(* PLC project WEEE_PLCs, Sconosciuto Senza_nome 1 *)
(* stored: creationDateTime 2024-08-18T12:18:40, modificationDateTime 2025-04-19T20:38:53 *)

TYPE STATUSES : (SHUT, OK, DANGER);
END_TYPE

TYPE FUNCTIONALITIES : (CONTROLLER, SEPARATOR);
END_TYPE

TYPE PLATFORM : STRUCT
  ID : INT;
  SHUTTED : BOOL;
  PC : REAL;
  SETTING : SETTINGS;
  STATUS : STATUSES;
  DIRECTION : DIRECTIONS;
  MATERIAL : MATERIALS;
END_STRUCT;
END_TYPE

TYPE SETTINGS : (AUTO, MANUAL);
END_TYPE

TYPE DIRECTIONS : (FORWARD, BACKWARD);
END_TYPE

TYPE WEIGHTS : (L, M, H);
END_TYPE

TYPE MATERIALS : (STEEL, COPPER, GOLD, CLAY, STONE);
END_TYPE

TYPE SHREADER : STRUCT
  ID : INT;
  PC : REAL;
  SETTING : SETTINGS;
  STATUS : STATUSES;
  WEIGHT : WEIGHTS;
END_STRUCT;
END_TYPE

FUNCTION_BLOCK PLATFORM_FB
  VAR_INPUT
    SHUTTED_IN : BOOL;
    SETTING_IN : INT;
    STATUS_IN : INT;
    PLATFORM_IN : PLATFORM;
  END_VAR
  VAR_OUTPUT
    STATUS_OUT : INT;
    PLATFORM_OUT : PLATFORM;
  END_VAR

            (*PLATFORM REMOTE CONFIGURATION*)
CASE SETTING_IN OF
  0: PLATFORM_IN.SETTING := MANUAL;
  1: PLATFORM_IN.SETTING := AUTO;
END_CASE;

(*SET PC BASED ON STATUS*)
IF SHUTTED_IN THEN
  PLATFORM_OUT.PC := 0.0;
  RETURN;
ELSE
  PLATFORM_OUT.PC := 3.5;
END_IF;

(*SET STATUS TO DANGER IF SOMETHING IS NOT NORMAL*)
IF PLATFORM_IN.PC >= 10.0 THEN
  PLATFORM_OUT.STATUS := DANGER;
ELSE
  PLATFORM_OUT.STATUS := OK;
END_IF;

(*UPDATE STATUS FOR MODBUS*)
CASE PLATFORM_OUT.STATUS OF
  OK: STATUS_OUT := 0;
  DANGER: STATUS_OUT := 1;
END_CASE;




          
END_FUNCTION_BLOCK

PROGRAM ClensePlc
  VAR
    C_ID : INT := 4;
    C_SHUTTED : BOOL;
    C_PILOT_STATUS : INT;
    C_PILOT_FUNC : INT;
    C_PC_INT : INT;
    C_STATUS : STATUSES;
    C_FUNC : FUNCTIONALITIES := CONTROLLER;
    C_PC_REAL : REAL := 0.0;
    C_WASTE_FB : PLATFORM_FB;
    C_WASTE : PLATFORM;
    C_WASTE_ID : INT := 8;
    C_WASTE_PC : REAL := 0.0;
    C_WASTE_SETTING : INT;
    C_WASTE_STATUS : INT;
    C_WASTE_DIRECTION : INT;
    C_WASTE_MATERIAL : INT;
  END_VAR
  VAR_EXTERNAL
    DENSITIES : ARRAY[0..2] OF PLATFORM;
  END_VAR
  VAR
    C_DENS_H_FB : PLATFORM_FB;
  END_VAR
  VAR_EXTERNAL
    DENS_H : PLATFORM;
    DENS_H_ID : INT;
    DENS_H_PC : REAL;
    DENS_H_SETTING : INT;
    DENS_H_STATUS : INT;
    DENS_H_DIRECTION : INT;
    DENS_H_MATERIAL : INT;
  END_VAR
  VAR
    C_DENS_M_FB : PLATFORM_FB;
  END_VAR
  VAR_EXTERNAL
    DENS_M : PLATFORM;
    DENS_M_ID : INT;
    DENS_M_PC : REAL;
    DENS_M_SETTING : INT;
    DENS_M_STATUS : INT;
    DENS_M_DIRECTION : INT;
    DENS_M_MATERIAL : INT;
  END_VAR
  VAR
    C_DENS_L_FB : PLATFORM_FB;
  END_VAR
  VAR_EXTERNAL
    DENS_L : PLATFORM;
    DENS_L_ID : INT;
    DENS_L_PC : REAL;
    DENS_L_SETTING : INT;
    DENS_L_STATUS : INT;
    DENS_L_DIRECTION : INT;
    DENS_L_MATERIAL : INT;
  END_VAR

            (*Define logic to assign enum value when receiving a command through modbus*)


(*Make the changes needed inside the function
C_WASTE_FB(
     IN := C_WASTE,
     OUT => C_WASTE);
*)

(*Update the variables with the new ones*)
C_WASTE_PC := C_WASTE.PC;

(*Set C_STATUS based on remote input*)


(*logic for functionality status*)



          
END_PROGRAM

PROGRAM DensityPlc
  VAR
    D_ID AT %QW3 : INT := 3;
  END_VAR
  VAR
    D_PC : REAL := 0.0;
    D_STATUS : STATUSES;
    D_PILOT_STATUS : INT;
    D_FUNC : FUNCTIONALITIES := SEPARATOR;
    D_GRIST_FB : PLATFORM_FB;
    D_GRIST : PLATFORM;
    D_GRIST_ID : INT := 20;
    D_GRIST_PC : REAL := 0.0;
    D_GRIST_SETTING : INT;
    D_GRIST_STATUS : INT;
    D_GRIST_DIRECTION : INT;
    D_GRIST_MATERIAL : INT;
  END_VAR
  VAR_EXTERNAL
    DENSITIES : ARRAY[0..2] OF PLATFORM;
  END_VAR
  VAR
    D_DENS_H_FB : PLATFORM_FB;
  END_VAR
  VAR_EXTERNAL
    DENS_H : PLATFORM;
    DENS_H_ID : INT;
    DENS_H_PC : REAL;
    DENS_H_SETTING : INT;
    DENS_H_STATUS : INT;
    DENS_H_DIRECTION : INT;
    DENS_H_MATERIAL : INT;
  END_VAR
  VAR
    D_DENS_M_FB : PLATFORM_FB;
  END_VAR
  VAR_EXTERNAL
    DENS_M : PLATFORM;
    DENS_M_ID : INT;
    DENS_M_PC : REAL;
    DENS_M_SETTING : INT;
    DENS_M_STATUS : INT;
    DENS_M_DIRECTION : INT;
    DENS_M_MATERIAL : INT;
  END_VAR
  VAR
    D_DENS_L_FB : PLATFORM_FB;
  END_VAR
  VAR_EXTERNAL
    DENS_L : PLATFORM;
    DENS_L_ID : INT;
    DENS_L_PC : REAL;
    DENS_L_SETTING : INT;
    DENS_L_STATUS : INT;
    DENS_L_DIRECTION : INT;
    DENS_L_MATERIAL : INT;
  END_VAR

            D_ID := 3;


          
END_PROGRAM

FUNCTION_BLOCK SHREADER_FB
  VAR_INPUT
    IN : SHREADER;
  END_VAR
  VAR_OUTPUT
    OUT : SHREADER;
  END_VAR

            OUT.ID := 3;


          
END_FUNCTION_BLOCK

PROGRAM ShreaderPlc
  VAR
    S_ID : INT := 2;
    S_PC : REAL := 0.0;
    S_STATUS : STATUSES;
    S_PILOT_STATUS : INT;
    S_FUNCTION : FUNCTIONALITIES := CONTROLLER;
    S_PILOT_FUNCTION : INT;
    S_SHREADER_FB : SHREADER_FB;
    S_SHREADER : SHREADER;
    S_SHREADER_ID : INT;
    S_SHREADER_PC : REAL := 0.0;
    S_SHREADER_SETTING : INT;
    S_SHREADER_STATUS : INT;
    S_SHREADER_WEIGHT : INT;
  END_VAR

            S_ID := 2;


          
END_PROGRAM

FUNCTION ShutPlcComponents : STATUSES
  VAR_OUTPUT
    PLC_PC : REAL;
    PLATFORM1_PC : REAL;
    PLATFORM2_PC : REAL;
    PLATFORM3_PC : REAL;
  END_VAR

            PLC_PC := 0.0;
PLATFORM1_PC := 0.0;
PLATFORM2_PC := 0.0;
PLATFORM3_PC := 0.0;

SHUTPLCCOMPONENTS := SHUT;

          
END_FUNCTION

PROGRAM WeightPlc
  VAR
    W_ID AT %QW1 : INT := 1;
    W_OPENED AT %QX0.0 : BOOL := 0;
  END_VAR
  VAR
    W_PC : REAL := 0.0;
  END_VAR
  VAR
    W_PC_INT AT %QW100 : INT := 0;
  END_VAR
  VAR
    W_STATUS : STATUSES;
  END_VAR
  VAR
    W_PILOT_STATUS AT %QW110 : INT := 0;
    W_CURRENT_STATUS AT %QW101 : INT := 0;
  END_VAR
  VAR
    W_FUNC : FUNCTIONALITIES := SEPARATOR;
  END_VAR
  VAR
    W_PILOT_FUNC AT %QW111 : INT := 1;
  END_VAR
  VAR
    WEIGHT_FB : PLATFORM_FB;
    WEIGHT_H : PLATFORM;
  END_VAR
  VAR
    WEIGHT_H_ID AT %QW102 : INT := 3;
  END_VAR
  VAR
    WEIGHT_H_SHUTTED : BOOL;
  END_VAR
  VAR
    WEIGHT_H_PC_INT AT %QW103 : INT := 0;
    WEIGHT_H_SETTING AT %QW112 : INT;
    WEIGHT_H_STATUS AT %QW113 : INT := 0;
    WEIGHT_H_DIRECTION AT %QW114 : INT;
    WEIGHT_H_MATERIAL AT %QW115 : INT;
  END_VAR
  VAR
    WEIGHT_M : PLATFORM;
  END_VAR
  VAR
    WEIGHT_M_ID AT %QW104 : INT := 2;
  END_VAR
  VAR
    WEIGHT_M_SHUTTED : BOOL;
  END_VAR
  VAR
    WEIGHT_M_PC_INT AT %QW105 : INT := 0;
    WEIGHT_M_SETTING AT %QW116 : INT;
    WEIGHT_M_STATUS AT %QW117 : INT;
    WEIGHT_M_DIRECTION AT %QW118 : INT;
    WEIGHT_M_MATERIAL AT %QW119 : INT;
  END_VAR
  VAR
    WEIGHT_L : PLATFORM;
  END_VAR
  VAR
    WEIGHT_L_ID AT %QW106 : INT := 1;
  END_VAR
  VAR
    WEIGHT_L_SHUTTED : BOOL;
  END_VAR
  VAR
    WEIGHT_L_PC_INT AT %QW107 : INT := 0;
    WEIGHT_L_SETTING AT %QW130 : INT;
    WEIGHT_L_STATUS AT %QW131 : INT;
    WEIGHT_L_DIRECTION AT %QW132 : INT;
    WEIGHT_L_MATERIAL AT %QW133 : INT;
  END_VAR

            (*COMPUTE PC FOR THIS PLC*)
(*NO NEED TO REMEMBER TO CONVERT REAL TO INT*)
W_PC_INT := REAL_TO_INT(W_PC * 10.0);
WEIGHT_H_PC_INT := REAL_TO_INT(WEIGHT_H.PC * 10.0);
WEIGHT_M_PC_INT := REAL_TO_INT(WEIGHT_M.PC * 10.0);
WEIGHT_L_PC_INT := REAL_TO_INT(WEIGHT_L.PC * 10.0);


(*WEIGHT PLC REMOTE CONFIGURATION*)

CASE W_PILOT_FUNC OF
  0: W_FUNC := CONTROLLER;
  1: W_FUNC := SEPARATOR;
END_CASE;

(*PLC VARIABLES SET*)
(*NORMALY OPEN IS THE SAFETY APPROACH IN A REAL WORLD SCENARIO*)
IF NOT W_OPENED THEN
  W_STATUS := ShutPlcComponents(
    PLC_PC => W_PC,
    PLATFORM1_PC => WEIGHT_H.PC,
    PLATFORM2_PC => WEIGHT_M.PC,
    PLATFORM3_PC => WEIGHT_L.PC);
    (*CLOSE EVERYTHING ATTACHED TO THIS PLC*)
ELSE
  W_PC := 1.5;
  W_STATUS := OK;
END_IF;

(*CHECK PLC STATUS BASED ON PC*)
IF W_PC >= 8.0 THEN (*MAYBE USE A GLOBAL VARIABLE FOR THE PC LIMIT...*)
  W_STATUS := DANGER;
END_IF;

(*MAP STATUS DATA TYPE WITH A UNIQUE NUMBER*)
CASE W_STATUS OF
  SHUT: W_CURRENT_STATUS := 0;
  OK: W_CURRENT_STATUS := 1;
  DANGER: W_CURRENT_STATUS := 2;
END_CASE;

(*CONTROL PLATFORMS ATTACHED TO THIS PLC*)
WEIGHT_FB(
     SETTING_IN := WEIGHT_H_SETTING,
     STATUS_IN := WEIGHT_H_STATUS,
     PLATFORM_IN := WEIGHT_H,
     STATUS_OUT => WEIGHT_H_STATUS,
     PLATFORM_OUT => WEIGHT_H);

WEIGHT_FB(
     SETTING_IN := WEIGHT_M_SETTING,
     STATUS_IN := WEIGHT_M_STATUS,
     PLATFORM_IN := WEIGHT_M,
     STATUS_OUT => WEIGHT_M_STATUS,
     PLATFORM_OUT => WEIGHT_M);

WEIGHT_FB(
     SETTING_IN := WEIGHT_L_SETTING,
     STATUS_IN := WEIGHT_L_STATUS,
     PLATFORM_IN := WEIGHT_L,
     STATUS_OUT => WEIGHT_L_STATUS,
     PLATFORM_OUT => WEIGHT_L);















          
END_PROGRAM

CONFIGURATION Config0
  RESOURCE Res0 ON PLC
    VAR_GLOBAL
      DENSITIES : ARRAY[0..2] OF PLATFORM;
      DENS_H : PLATFORM;
      DENS_H_ID : INT := 7;
      DENS_H_PC : REAL := 0.0;
      DENS_H_SETTING : INT;
      DENS_H_STATUS : INT;
      DENS_H_DIRECTION : INT;
      DENS_H_MATERIAL : INT;
      DENS_M : PLATFORM;
      DENS_M_ID : INT := 6;
      DENS_M_PC : REAL := 0.0;
      DENS_M_SETTING : INT;
      DENS_M_STATUS : INT;
      DENS_M_DIRECTION : INT;
      DENS_M_MATERIAL : INT;
      DENS_L : PLATFORM;
      DENS_L_ID : INT := 5;
      DENS_L_PC : REAL := 0.0;
      DENS_L_SETTING : INT;
      DENS_L_STATUS : INT;
      DENS_L_DIRECTION : INT;
      DENS_L_MATERIAL : INT;
    END_VAR
    TASK task0(INTERVAL := T#20ms, PRIORITY := 0);
    PROGRAM instance0 WITH task0 : WeightPlc;
  END_RESOURCE
END_CONFIGURATION
